% RSLogix 500 project I2P JOB 12B - TYLER_VOGT.RSS, saved by version 10.00.00.00 %
PROJECT "MLO2B"    % processor: Bul.1763 MicroLogix 1100 Series B %

PROGRAM FILES
  LAD 2   12 rungs

DATA FILES
  O0 OUTPUT  4 elements
  I1 INPUT  6 elements
  S2 STATUS  66 elements
  B3 BINARY  1 elements
  T4 TIMER  2 elements
  C5 COUNTER  1 elements
  R6 CONTROL  1 elements
  N7 INTEGER  1 elements
  F8 FLOAT  1 elements

LADDER 2
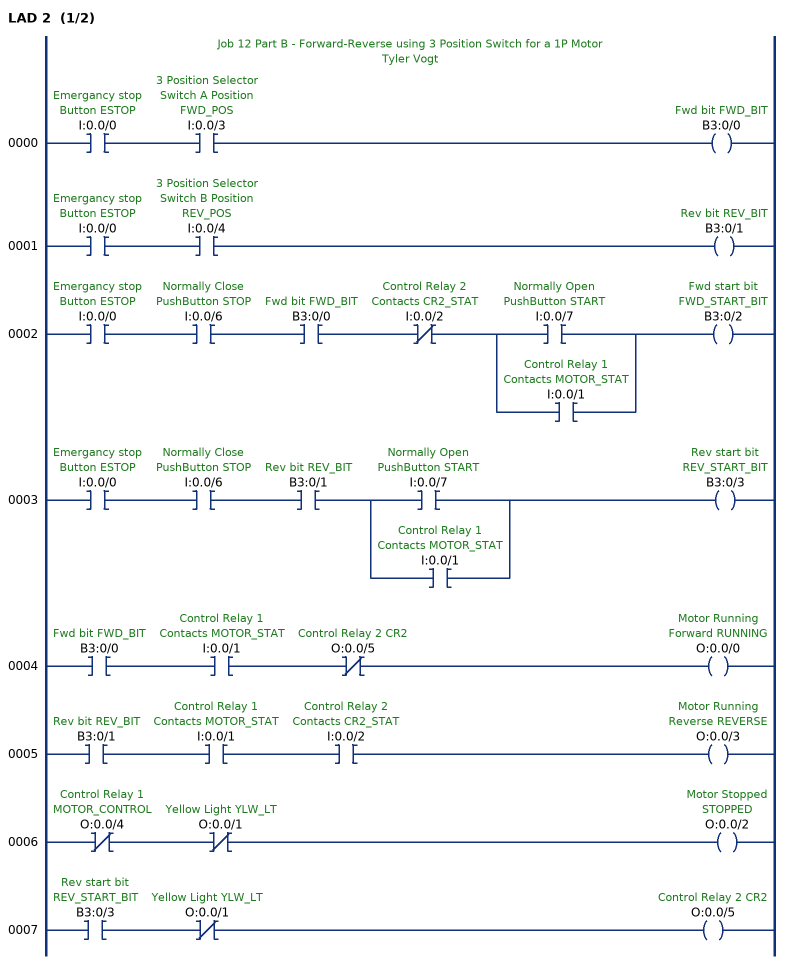
% Rung: 0 %
% Job 12 Part B - Forward-Reverse using 3 Position Switch for a 1P Motor
% Tyler Vogt %
SOR XIC I:0.0/0 XIC I:0.0/3 OTE B3:0/0 EOR
%   I:0.0/0  ESTOP  "Emergancy stop Button" %
%   I:0.0/3  FWD_POS  "3 Position Selector Switch A Position" %
%   B3:0/0  FWD_BIT  "Fwd bit" %
% Rung: 1 %
SOR XIC I:0.0/0 XIC I:0.0/4 OTE B3:0/1 EOR
%   I:0.0/0  ESTOP  "Emergancy stop Button" %
%   I:0.0/4  REV_POS  "3 Position Selector Switch B Position" %
%   B3:0/1  REV_BIT  "Rev bit" %
% Rung: 2 %
SOR XIC I:0.0/0 XIC I:0.0/6 XIC B3:0/0 XIO I:0.0/2 BST XIC I:0.0/7 NXB XIC I:0.0/1 BND OTE B3:0/2 EOR
%   I:0.0/0  ESTOP  "Emergancy stop Button" %
%   I:0.0/6  STOP  "Normally Close PushButton" %
%   B3:0/0  FWD_BIT  "Fwd bit" %
%   I:0.0/2  CR2_STAT  "Control Relay 2 Contacts" %
%   I:0.0/7  START  "Normally Open PushButton" %
%   I:0.0/1  MOTOR_STAT  "Control Relay 1 Contacts" %
%   B3:0/2  FWD_START_BIT  "Fwd start bit" %
% Rung: 3 %
SOR XIC I:0.0/0 XIC I:0.0/6 XIC B3:0/1 BST XIC I:0.0/7 NXB XIC I:0.0/1 BND OTE B3:0/3 EOR
%   I:0.0/0  ESTOP  "Emergancy stop Button" %
%   I:0.0/6  STOP  "Normally Close PushButton" %
%   B3:0/1  REV_BIT  "Rev bit" %
%   I:0.0/7  START  "Normally Open PushButton" %
%   I:0.0/1  MOTOR_STAT  "Control Relay 1 Contacts" %
%   B3:0/3  REV_START_BIT  "Rev start bit" %
% Rung: 4 %
SOR XIC B3:0/0 XIC I:0.0/1 XIO O:0.0/5 OTE O:0.0/0 EOR
%   B3:0/0  FWD_BIT  "Fwd bit" %
%   I:0.0/1  MOTOR_STAT  "Control Relay 1 Contacts" %
%   O:0.0/5  CR2  "Control Relay 2" %
%   O:0.0/0  RUNNING  "Motor Running Forward" %
% Rung: 5 %
SOR XIC B3:0/1 XIC I:0.0/1 XIC I:0.0/2 OTE O:0.0/3 EOR
%   B3:0/1  REV_BIT  "Rev bit" %
%   I:0.0/1  MOTOR_STAT  "Control Relay 1 Contacts" %
%   I:0.0/2  CR2_STAT  "Control Relay 2 Contacts" %
%   O:0.0/3  REVERSE  "Motor Running Reverse" %
% Rung: 6 %
SOR XIO O:0.0/4 XIO O:0.0/1 OTE O:0.0/2 EOR
%   O:0.0/4  MOTOR_CONTROL  "Control Relay 1" %
%   O:0.0/1  YLW_LT  "Yellow Light" %
%   O:0.0/2  STOPPED  "Motor Stopped" %
% Rung: 7 %
SOR XIC B3:0/3 XIO O:0.0/1 OTE O:0.0/5 EOR
%   B3:0/3  REV_START_BIT  "Rev start bit" %
%   O:0.0/1  YLW_LT  "Yellow Light" %
%   O:0.0/5  CR2  "Control Relay 2" %

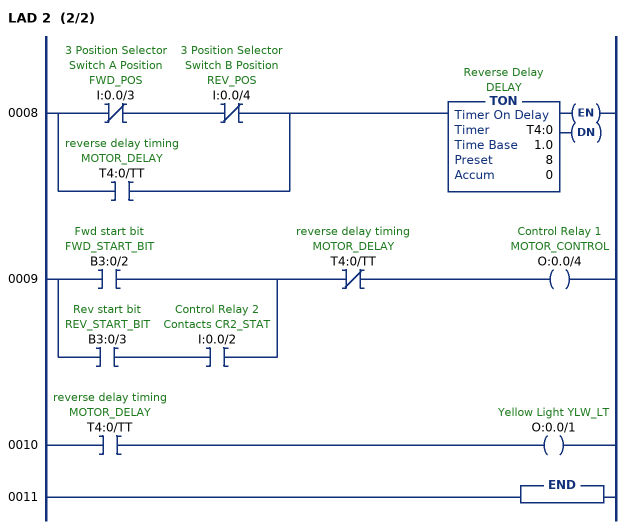
% Rung: 8 %
SOR BST XIO I:0.0/3 XIO I:0.0/4 NXB XIC T4:0/TT BND TON T4:0 1.0 8 0 EOR
%   I:0.0/3  FWD_POS  "3 Position Selector Switch A Position" %
%   I:0.0/4  REV_POS  "3 Position Selector Switch B Position" %
%   T4:0/TT  MOTOR_DELAY  "reverse delay timing" %
%   T4:0  DELAY  "Reverse Delay" %
% Rung: 9 %
SOR BST XIC B3:0/2 NXB XIC B3:0/3 XIC I:0.0/2 BND XIO T4:0/TT OTE O:0.0/4 EOR
%   B3:0/2  FWD_START_BIT  "Fwd start bit" %
%   B3:0/3  REV_START_BIT  "Rev start bit" %
%   I:0.0/2  CR2_STAT  "Control Relay 2 Contacts" %
%   T4:0/TT  MOTOR_DELAY  "reverse delay timing" %
%   O:0.0/4  MOTOR_CONTROL  "Control Relay 1" %
% Rung: 10 %
SOR XIC T4:0/TT OTE O:0.0/1 EOR
%   T4:0/TT  MOTOR_DELAY  "reverse delay timing" %
%   O:0.0/1  YLW_LT  "Yellow Light" %
% Rung: 11 %
SOR END EOR

OTHER DOCUMENTED ADDRESSES
  I:0.0/5  RUN_JOG  "2 Position Selector Switch A Position"
  I:0.0/8  JOG  "Normally Open PushButton"
  T4:1  REV_DELAY  "Forward Delay"
  T4:1/TT  REV_DELAY_TIMING  "Forward timing delay"

DATA TABLE (non-zero values as saved)
DATA T4
% .PRE .ACC %
% T4:0 % 8 0
% T4:1 % 8 0
